FUNCTION_BLOCK TwoConCtlRingToken (* Composite Function Block Type *)
  (* Standard: 61499-2 *)
  (* Version 0.2, 2003-12-05, JHC, Rockwell Automation, Renamed from NEWCOMPFB. *)
  (* Version 0.1, 2002-01-08, JHC, Rockwell Automation, Added DLY FB as example. *)
  (* Version 0.0, 2000-05-27, JHC, Rockwell Automation *)
  (* Compiler header: package fb.rt.cs725; *)
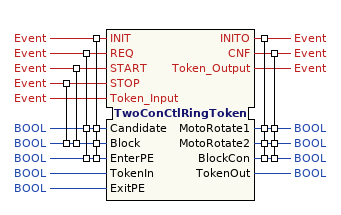
  EVENT_INPUT
    INIT WITH Candidate, Block, EnterPE; (* Initialization Request *)
    REQ WITH Candidate, EnterPE; (* Normal Execution Request *)
    START WITH Block;
    STOP WITH Block;
    Token_Input;
  END_EVENT
  EVENT_OUTPUT
    INITO WITH MotoRotate1, MotoRotate2, BlockCon; (* Initialization Confirm *)
    CNF WITH MotoRotate1, MotoRotate2, BlockCon; (* Execution Confirmation *)
    Token_Output;
  END_EVENT
  VAR_INPUT
    Candidate : BOOL;
    Block : BOOL;
    EnterPE : BOOL;
    TokenIn : BOOL;
    ExitPE : BOOL;
  END_VAR
  VAR_OUTPUT
    MotoRotate1 : BOOL;
    MotoRotate2 : BOOL;
    BlockCon : BOOL;
    TokenOut : BOOL;
  END_VAR
  FBS
    FC11 : ConveyorCTL(PE := 0, Block := 0, Candidate := 0);
    RingToken : RingToken;
  END_FBS
  EVENT_CONNECTIONS
    INIT TO FC11.INIT;
    REQ TO FC11.REQ;
    RingToken.STOP TO FC11.CAS_STOP;
    RingToken.START TO FC11.CAS_START;
    RingToken.INITO TO INITO;
    FC11.INITO TO RingToken.INIT;
    REQ TO RingToken.REQ;
    STOP TO RingToken.CAS_STOP;
    START TO RingToken.CAS_START;
    Token_Input TO RingToken.Token_Input;
    RingToken.Token_Output TO Token_Output;
  END_CONNECTIONS
  DATA_CONNECTIONS
    FC11.MotoRotate TO MotoRotate1;
    RingToken.MotoRotate TO MotoRotate2;
    RingToken.BlockCon TO BlockCon;
    RingToken.TokenOut TO TokenOut;
    EnterPE TO RingToken.EnterPE;
    Block TO RingToken.Block;
    Candidate TO RingToken.Candidate;
    TokenIn TO RingToken.TokenIn;
    ExitPE TO RingToken.ExitPE;
  END_CONNECTIONS
END_FUNCTION_BLOCK
